{attribute addProperty BoxType "EP8309-0022-0021"}
{attribute addProperty Id "Undervoltage_UsAT %I*BOOL811Undervoltage_UpAT %I*BOOL812"}
{attribute addProperty CRC "2794300337"}
{attribute addProperty SizeInBites "16"}
{attribute addProperty SizeInBytes "2"}
TYPE DEV_Inputs_A68DA3B1 :
STRUCT
	{attribute addProperty Name "Undervoltage_Us"}
	Undervoltage_Us AT %I* : BOOL;
	{attribute addProperty Name "Undervoltage_Up"}
	Undervoltage_Up AT %I* : BOOL;
END_STRUCT
END_TYPE

(* stored: Version 1.2.0.0, ProductVersion 3.1.4024.9
   DUT DEV_Inputs_A68DA3B1: Id {325abbae-3856-47ee-9635-a43b7a70292e} *)
